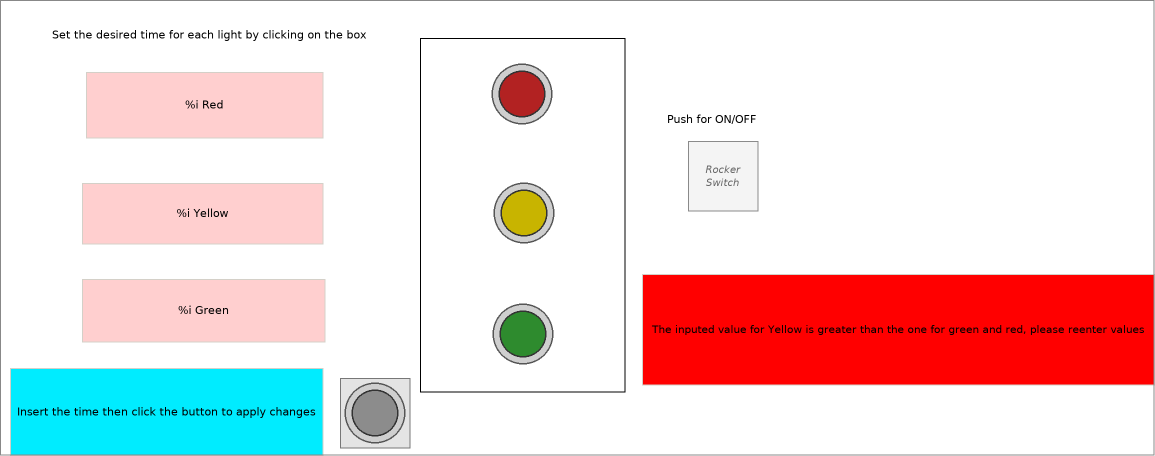
VISUALIZATION Visualization  // 1155x456
    Rectangle (420,38 205x354)
    Lamp1 (487,59 70x70), variable: TrafficLight.bRedLight, style: Lamp-Lamp1-Red
    Lamp1 (489,178 70x70), variable: TrafficLight.bYellowLight, style: Lamp-Lamp1-Yellow
    Lamp1 (488,299 70x70), variable: TrafficLight.bGreenLight, style: Lamp-Lamp1-Green
    Label (34,20 351x30), "Set the desired time for each light by clicking on the box"
    Textfield (86,72 237x66), "%i Red", text variable: TrafficLight.iRedColor
        OnMouseDown: write the text variable via Default
    Textfield (82,183 241x61), "%i Yellow", text variable: TrafficLight.iYellowColor
        OnMouseDown: write the text variable via Default
    Textfield (82,279 243x63), "%i Green", text variable: TrafficLight.iGreenColor
        OnMouseDown: write the text variable via Default
    RockerSwitch (688,141 70x70), variable: TrafficLight.bTurnOn, behaviour: TOGGLE, style: Switch-RockerSwitch-Red
    Label (659,98 106x43), "Push for ON/OFF"
    Textfield (642,274 513x111), "The inputed value for Yellow is greater than the one for green and red, please reenter values", invisible if: TrafficLight.bTextError
    PushSwitch (340,378 70x70), variable: TrafficLight.bTempActive, behaviour: TAP, style: Switch-PushSwitch-Gray
    Textfield (10,368 313x88), "Insert the time then click the button to apply changes"
END_VISUALIZATION

(* stored: Version 1.1.0.1, ProductVersion 3.1.4024.12
   Visu Visualization: Id {b6933371-4b8d-4c31-a69e-acb393bb7aeb} *)
